// SIMATIC S7-200 project (STEP 7-Micro/WIN), CPU 224XP CN REL 02.01

SYMBOL_TABLE 用户定义1
ADD1             VW1
ADD2             VW3
ADD3             VW5
ADDANS           VW7
MODDONE          M0.0
MODSDONE         M0.1
MODERR           MB1
MODSERR          MB3
END_SYMBOL_TABLE

ORGANIZATION_BLOCK 主程序:OB1
TITLE=程序注释
BEGIN
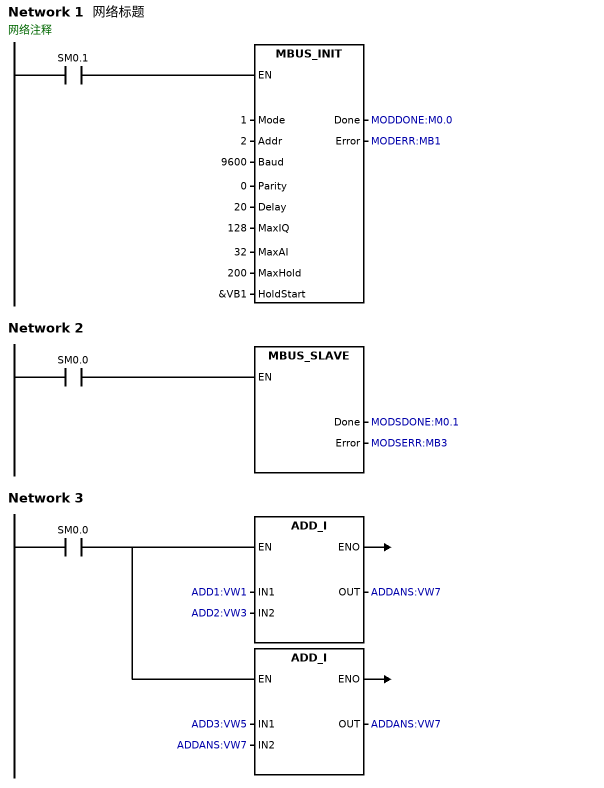
Network 1 // 网络标题
// 网络注释
LD     SM0.1
CALL   MBUS_INIT:SBR1, 1, 2, 9600, 0, 20, 128, 32, 200, &VB1, MODDONE:M0.0, MODERR:MB1
Network 2
LD     SM0.0
CALL   MBUS_SLAVE:SBR2, MODSDONE:M0.1, MODSERR:MB3
Network 3
LD     SM0.0
MOVW   ADD1:VW1, ADDANS:VW7
+I     ADD2:VW3, ADDANS:VW7
+I     ADD3:VW5, ADDANS:VW7
END_ORGANIZATION_BLOCK

// SBR1: protected block, not included

// SBR2: protected block, not included

// SBR3: protected block, not included
